# B&R Automation Studio project lektion_VI_agdp
Automation Studio 4.8.2.72


## Logical view

### Program Logical/Opg1 (IEC)

#### Variables.var
```iecst
VAR
	A : USINT;
	shift : BOOL;
	i : USINT;
END_VAR
```

### Program Logical/Opg2 (IEC)

#### Main.st
```iecst
PROGRAM _INIT
	(* Insert code here *)
	array[0] := TRUE;
	shift := TRUE;

END_PROGRAM

PROGRAM _CYCLIC
	(* Insert code here *)
	IF shift THEN
		tmp := array[0];
		array[0] := array[1];
		array[1] := array[2];
		array[2] := array[3];
		array[3] := array[4];
		array[4] := array[5];
		array[5] := array[6];
		array[6] := array[7];
		array[7] := array[8];
		array[8] := array[9];
		array[9] := array[10];
		array[10] := array[11];
		array[11] := array[12];
		array[12] := array[13];
		array[13] := array[14];
		array[14] := array[15];
		array[15] := tmp;
	END_IF;

END_PROGRAM

PROGRAM _EXIT
	(* Insert code here *)

END_PROGRAM
```

### Program Logical/Program

#### Main.st
```iecst
PROGRAM _INIT
	(* Insert code here *)
	VAR
		aBitshifting : ARRAY[0..15] OF BOOL;
	END_VAR

	aBitshifting[15] := true;

END_PROGRAM

PROGRAM _CYCLIC
	(* Insert code here *)
	A := A + 1;

END_PROGRAM

PROGRAM _EXIT
	(* Insert code here *)

END_PROGRAM
```

Listed in the project but not available here: Logical/Global.typ, Logical/Global.var, Logical/Libraries
